Staubli VAL3: adept04.dtx


